// TIA Portal V15.1 export
// export: Created 2024-06-21T08:40:43.1871173Z, ExportSetting WithDefaults, DisplayName Totally Integrated Automation Portal, DisplayVersion V15.1 Update 5, DisplayName TIA Portal Openness, DisplayVersion V15.1 Update 5, DisplayName SINAMICS Startdrive Advanced, DisplayVersion V15.1, DisplayName G130, G150, S120, S150, SINAMICS MV, S210, DisplayVersion V15.1, DisplayName G110M, G120, G120C, G120D, G120P, DisplayVersion V15.1, DisplayName STEP 7 Professional, DisplayVersion V15.1 Update 5, DisplayName STEP 7 Safety, DisplayVersion V15.1, DisplayName WinCC Professional, DisplayVersion V15.1 Update 5, DisplayName SIMATIC Visualization Architect, DisplayVersion V15.1
DATA_BLOCK "_209220ZM01AlarmsCompare"   // DB132
{ S7_Optimized_Access := 'FALSE' }
AUTHOR : VCC
FAMILY : ALARM
NAME : ALARMDB
VERSION : 0.1
// stored: AutoNumber false, DBAccessibleFromOPCUA true, IsOnlyStoredInLoadMemory false, IsWriteProtectedInAS false
   VAR RETAIN
      VDHeaderLength { ExternalAccessible := 'False'; ExternalVisible := 'False'; ExternalWritable := 'False'} : Word;   // VD Header length of the DB
      VDHeaderDBNumber { ExternalAccessible := 'False'; ExternalVisible := 'False'; ExternalWritable := 'False'} : Word;   // VD Header DB Number
      "209220ZM01_AW1" { ExternalAccessible := 'False'; ExternalVisible := 'False'; ExternalWritable := 'False'} : DWord;   // Alarm Word
      "209220ZMS011Modes_AW1" { ExternalAccessible := 'False'; ExternalVisible := 'False'; ExternalWritable := 'False'} : DWord;   // Alarm Word
      "209220ZMS012Modes_AW1" { ExternalAccessible := 'False'; ExternalVisible := 'False'; ExternalWritable := 'False'} : DWord;   // Alarm Word
      "209220ZMS013Modes_AW1" { ExternalAccessible := 'False'; ExternalVisible := 'False'; ExternalWritable := 'False'} : DWord;   // Alarm Word
      "209220ZMS011ProdMode_AW1" { ExternalAccessible := 'False'; ExternalVisible := 'False'; ExternalWritable := 'False'} : DWord;   // Alarm Word
      "209220ZMS012ProdMode_AW1" { ExternalAccessible := 'False'; ExternalVisible := 'False'; ExternalWritable := 'False'} : DWord;   // Alarm Word
      "209220ZMS013ProdMode_AW1" { ExternalAccessible := 'False'; ExternalVisible := 'False'; ExternalWritable := 'False'} : DWord;   // Alarm Word
      "209220ZM01Orders_AW1" { ExternalAccessible := 'False'; ExternalVisible := 'False'; ExternalWritable := 'False'} : DWord;   // Alarm Word
      "209220ZM01DataHandling_AW1" { ExternalAccessible := 'False'; ExternalVisible := 'False'; ExternalWritable := 'False'} : DWord;   // Alarm Word
      "209220ZM01Andon_AW1" { ExternalAccessible := 'False'; ExternalVisible := 'False'; ExternalWritable := 'False'} : DWord;   // Alarm Word
      "209220ZM01NCB01TagSequence_AW1" { ExternalAccessible := 'False'; ExternalVisible := 'False'; ExternalWritable := 'False'} : DWord;   // Alarm Word
      "209220ZM01NCB02TagSequence_AW1" { ExternalAccessible := 'False'; ExternalVisible := 'False'; ExternalWritable := 'False'} : DWord;   // Alarm Word
      "209220ZM01CRClockStartStop_AW1" { ExternalAccessible := 'False'; ExternalVisible := 'False'; ExternalWritable := 'False'} : DWord;   // Alarm Word
      "209220CS22ProdSpeed_AW1" { ExternalAccessible := 'False'; ExternalVisible := 'False'; ExternalWritable := 'False'} : DWord;   // Alarm Word
      "209220CS22LineFeed_AW1" { ExternalAccessible := 'False'; ExternalVisible := 'False'; ExternalWritable := 'False'} : DWord;   // Alarm Word
      "209220CS22ProdStartStop_AW1" { ExternalAccessible := 'False'; ExternalVisible := 'False'; ExternalWritable := 'False'} : DWord;   // Alarm Word
      "209220CS22ShiftRegLine_AW1" { ExternalAccessible := 'False'; ExternalVisible := 'False'; ExternalWritable := 'False'} : DWord;   // Alarm Word
      "209220CHB21_AW1" { ExternalAccessible := 'False'; ExternalVisible := 'False'; ExternalWritable := 'False'} : DWord;   // Alarm Word
      "209220CR21_AW1" { ExternalAccessible := 'False'; ExternalVisible := 'False'; ExternalWritable := 'False'} : DWord;   // Alarm Word
      "209220CS22_AW1" { ExternalAccessible := 'False'; ExternalVisible := 'False'; ExternalWritable := 'False'} : DWord;   // Alarm Word
      "209220CR23_AW1" { ExternalAccessible := 'False'; ExternalVisible := 'False'; ExternalWritable := 'False'} : DWord;   // Alarm Word
      "209000AE01E3FS10CH1_AW1" { ExternalAccessible := 'False'; ExternalVisible := 'False'; ExternalWritable := 'False'} : DWord;   // Alarm Word
      "209000AE01E3FS10CH2_AW1" { ExternalAccessible := 'False'; ExternalVisible := 'False'; ExternalWritable := 'False'} : DWord;   // Alarm Word
      "209000AE01E3FS11CH1_AW1" { ExternalAccessible := 'False'; ExternalVisible := 'False'; ExternalWritable := 'False'} : DWord;   // Alarm Word
      "209000AE01E3FS11CH2_AW1" { ExternalAccessible := 'False'; ExternalVisible := 'False'; ExternalWritable := 'False'} : DWord;   // Alarm Word
      "209000AK02E3FS56CH1_AW1" { ExternalAccessible := 'False'; ExternalVisible := 'False'; ExternalWritable := 'False'} : DWord;   // Alarm Word
      "209000AK02E3FS200CH1_AW1" { ExternalAccessible := 'False'; ExternalVisible := 'False'; ExternalWritable := 'False'} : DWord;   // Alarm Word
      "209000AK02E3FS200CH2_AW1" { ExternalAccessible := 'False'; ExternalVisible := 'False'; ExternalWritable := 'False'} : DWord;   // Alarm Word
      "209000AK02E3FS201CH1_AW1" { ExternalAccessible := 'False'; ExternalVisible := 'False'; ExternalWritable := 'False'} : DWord;   // Alarm Word
      "209000AK02E3FS201CH2_AW1" { ExternalAccessible := 'False'; ExternalVisible := 'False'; ExternalWritable := 'False'} : DWord;   // Alarm Word
      "209000AK02E3FS202CH1_AW1" { ExternalAccessible := 'False'; ExternalVisible := 'False'; ExternalWritable := 'False'} : DWord;   // Alarm Word
      "209000AK02E3FS202CH2_AW1" { ExternalAccessible := 'False'; ExternalVisible := 'False'; ExternalWritable := 'False'} : DWord;   // Alarm Word
      "209000AK02E3FS203CH1_AW1" { ExternalAccessible := 'False'; ExternalVisible := 'False'; ExternalWritable := 'False'} : DWord;   // Alarm Word
      "209000AK02E3FS203CH2_AW1" { ExternalAccessible := 'False'; ExternalVisible := 'False'; ExternalWritable := 'False'} : DWord;   // Alarm Word
   END_VAR
BEGIN
END_DATA_BLOCK
